// TIA Portal V17 export
// export: Created 2023-03-06T02:05:26.0829886Z, ExportSetting WithDefaults, DisplayName Totally Integrated Automation Portal, DisplayVersion V17 Update 4, DisplayName TIA Portal Openness, DisplayVersion V17 Update 4, DisplayName TIA Portal Version Control Interface, DisplayVersion V17, DisplayName STEP 7 Professional, DisplayVersion V17 Update 4, DisplayName STEP 7 Safety, DisplayVersion V17, DisplayName WinCC Professional, DisplayVersion V17 Update 4
TYPE "BMS_BR"
// stored: IsFailsafeCompliant false
   STRUCT
      wWarn1 : Word;   // Warning_1
      wWarn2 : Word;   // Warning_2
      wWarn3 : Word;   // Warning_3
      wWarn4 : Word;   // Warning_4
      xKprechSt : Bool;   // Prech_Relay_Status
      xKposSt : Bool;   // Pos_Relay_Status
      xKnegSt : Bool;   // Neg_Relay_Status
      xBalSt : Bool;   // Balance_Status
      rVdcMeas : Real;   // Voltage
      rIdcMeas : Real;   // Current
      rSOCmeas : Real;   // SOC
      rSOHmeas : Real;   // SOH
      rVcellMaxMeas : Real;   // Max_Cell_Volt
      rVcellMinMeas : Real;   // Min_Cell_Volt
      rVcellAvgMeas : Real;   // Avg_Cell_Volt
      iTcellMaxMeas : Int;   // Max_Cell_Temp
      iTcellMinMeas : Int;   // Min_Cell_Temp
      iTcellAvgMeas : Int;   // Avg_Cell_Temp
      rIchaLim : Real;   // Max_Allowed_Ch_Curr
      rIdschLim : Real;   // Max_Allowed_Dh_Curr
      iVcellMaxPos : Int;   // Max_Cell_Volt_Pos Byte 0
      iVcellMinPos : Int;   // Max_Cell_Volt_Pos Byte 1
      iTcellMaxPos : Int;   // Min_Cell_Volt_Pos Byte 0
      iTcellMinPos : Int;   // Min_Cell_Volt_Pos Byte 1
      iVmodMaxPos : Int;   // Max_Cell_Temp_Pos Byte 0
      iVmodMinPos : Int;   // Max_Cell_Temp_Pos Byte 1
      iTmodMaxPos : Int;   // Min_Cell_Temp_Pos Byte 0
      iTmodMinPos : Int;   // Min_Cell_Temp_Pos Byte 1
      rVcellSumMeas : Real;   // Sum_Cell_Voltage
      iTrackInMeas : Int;   // Rack_Inlet_Temp
      iTrackOutMeas : Int;   // Rack_Outlet_Temp
      iTambMeas : Int;   // Environment_Temp
      xDoorSt : Bool;   // Door_State
      xFanSt : Bool;   // Fan_State
   END_STRUCT;
END_TYPE
